Universal Robots PolyScope program: VisionCognex.urp

Program VisionCognex (installation=VisionCognex directory=/programs createdIn=3.0.17779.0 lastSavedIn=5.9.1.1031110 robotSerialNumber=20195501059)
Calibrated DH parameters: a=[0.000146, -0.418764, -0.053981, 0.000058, -0.000023, 0]; d=[0.162545, 37.319448, -206.067439, 168.881546, 0.09955, 0.099464]; alpha=[1.57004, -0.001979, 0.002304, 1.570607, -1.57066, 0]; deltaTheta=[0, -0.174616, -1.258233, 1.432844, -0.000001, 0]
BeforeStart
  Call InitialData
  Call InitialPosition
  Call InitialConnect
Robot Program (runOnlyOnce=false)
  Call DoPrepare
  Call CallCameraSnap
  Call GetCameraData
  Call GoNewPosition
  Call ClearAllData
SubProgram -> InitialData
SubProgram -> InitialPosition
SubProgram -> InitialConnect
SubProgram -> DoPrepare
SubProgram -> CallCameraSnap
SubProgram -> GetCameraData
SubProgram -> GoNewPosition
SubProgram -> ClearAllData
SubProgram InitialData (keepSynchronizedWithDisk=false)
  'only need three parameters from camera,so the array length will be 4'
  TargetObject := [0,0,0,0,0]
  TargetX := 0
  TargetY := 0
  TargetRotation := 0
  TargetPercent := 0
  'the following variable defines how much mm 1 pixel equals'
  PixelDistance := (0.09*0.001)
  RefObjectX := 199
  RefObjectY := 188
  Script: set_tool_voltage(24)
SubProgram InitialPosition (keepSynchronizedWithDisk=false)
  'Before we trigger the camera, we will go the zero point of the board'
  MoveJ speed 60 deg/s, acceleration 80 deg/s^2 (useActiveTCP=false) feature=Base
    Waypoint Prepare: TCP in base x=201.696 y=-681.245 z=177.165 mm, rx=-0.2909 ry=-3.1191 rz=-0.0205 rad; joints [95.679, -50.567, 83.407, -121.999, 269.63, -343.651] deg
  SuppressedNode
    MoveJ speed 60 deg/s, acceleration 80 deg/s^2 (useActiveTCP=false) feature=Base
      Waypoint BoradZeroPre: TCP in base x=-93.243 y=446.159 z=22.323 mm, rx=2.173 ry=2.2023 rz=-0.0207 rad; joints [116.026, -102.96, -125.452, -44.455, 89.644, -64.941] deg; TCP offset x=-10.197 y=-18.74 z=156.717 mm, rx=0.0017 ry=-0.0003 rz=0.007 rad
      PosZeroPre := get_target_tcp_pose()
      Waypoint BoardZeroPick: TCP in base x=-92.727 y=445.244 z=2.429 mm, rx=2.1728 ry=2.2021 rz=-0.0208 rad; joints [116.02, -105.4, -126.53, -40.936, 89.652, -64.959] deg; TCP offset x=-10.228 y=-18.656 z=156.723 mm, rx=0.0013 ry=-0.0004 rz=0.0071 rad
      PosZeroPick := get_target_tcp_pose()
  PosZeroPre := BoardZero
  PosZeroPick := BoardZeroTruely
SubProgram InitialConnect (keepSynchronizedWithDisk=false)
  Connected := False
  Loop While (checkContinuously=false) expression=Connected≟ False
    Connected := socket_open("192.168.0.251",3000,"socket0")
    Wait Sleep waitTime=0.5
SubProgram DoPrepare (keepSynchronizedWithDisk=false)
  'move the robot to a position and wait to pick object'
  MoveJ speed 60 deg/s, acceleration 80 deg/s^2 (useActiveTCP=false) feature=Base
    Waypoint Prepare: TCP in base x=201.696 y=-681.245 z=177.165 mm, rx=-0.2909 ry=-3.1191 rz=-0.0205 rad; joints [95.679, -50.567, 83.407, -121.999, 269.63, -343.651] deg
    Set DigitalOutput pin=tool_out[0]; digitalValue=0
    Popup Message (haltProgram=false message=Please put target object to a place inputType=Text)
SubProgram CallCameraSnap (keepSynchronizedWithDisk=false)
  'after we tell camera to take snapshot,we can make a stopwatch to see the responese time of the camera'
  Loop Counting (count=1) loopVariable(name=循环_1)
    Script: socket_send_string("r","socket0")
    Script: socket_send_byte(13,"socket0")
    Wait Sleep waitTime=0.01
SubProgram GetCameraData (keepSynchronizedWithDisk=false)
  'wait until the camare give me data'
  Loop While (checkContinuously=false) expression=TargetObject[0]≟0
    TargetObject := socket_read_ascii_float(4,"socket0")
    Wait Sleep waitTime=0.1
  'put the data into my own variable,remember the TargetObject[0] has stored the array length'
  TargetX := (TargetObject[1]-RefObjectX)*PixelDistance
  TargetY := (TargetObject[2]-RefObjectY)*PixelDistance
  TargetRotation := -d2r(TargetObject[3])
  TargetPercent := TargetObject[4]
  If TargetPercent≟0
    Popup Message (haltProgram=false message=Not find the pattern inputType=Text)
SubProgram GoNewPosition (keepSynchronizedWithDisk=false)
  'the most easy way will be use function pose_trans'
  AddPos := p[-TargetX,TargetY,0,0,0,TargetRotation]
  NewPosPre := pose_trans(PosZeroPre,AddPos)
  NewPosPick := pose_trans(PosZeroPick,AddPos)
  MoveL speed 250 mm/s, acceleration 1200 mm/s^2 (useActiveTCP=true) feature=Base
    Waypoint Waypoint (Variable): variable=NewPosPre
    Waypoint Waypoint (Variable): variable=NewPosPick
    Set DigitalOutput pin=tool_out[0]; digitalValue=1
    Wait Sleep waitTime=1
    Waypoint Waypoint (Variable): variable=NewPosPre
SubProgram ClearAllData (keepSynchronizedWithDisk=false)
  TargetObject := [0,0,0,0,0]
  Wait Sleep waitTime=0.01
